{attribute 'qualified_only'}
{attribute 'strict'}
TYPE EDisplayControlStep :
(
	Percent_0 := 0,
	Percent_25 := 1,
	Percent_50 := 2,
	Percent_75 := 3,
	Percent_100 := 4
);
END_TYPE

(* stored: Version 1.1.0.1, ProductVersion 3.1.4024.12
   DUT EDisplayControlStep: Id {12e5c99c-99e0-406f-bc10-32e2bc164870} *)
